// TIA Portal V15 export
FUNCTION "Preset_main" : Void   // FC30, SCL
{ S7_Optimized_Access := 'TRUE' }
VERSION : 0.1
// stored: AutoNumber true, IsIECCheckEnabled false, SetENOAutomatically False
   VAR_INPUT
      Value : "PresetValueType";
      Enable : "PresetEnableType";
   END_VAR
BEGIN
END_FUNCTION
